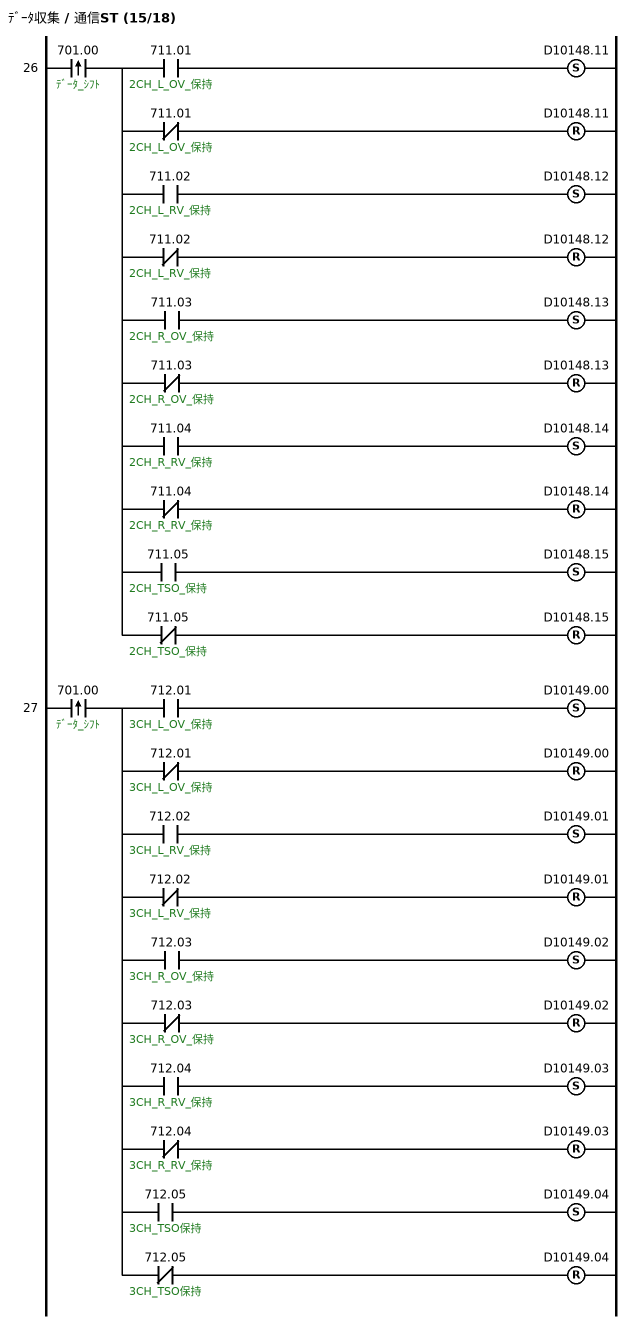
; [picture p216: ﾃﾞｰﾀ収集 / 通信ST, rungs 26-27]
; rung 26
@LD 701.00  ; ﾃﾞｰﾀ_ｼﾌﾄ
OUT TR0
AND 711.01  ; 2CH_L_OV_保持
SET D10148.11
LD TR0
ANDNOT 711.01  ; 2CH_L_OV_保持
RSET D10148.11
LD TR0
AND 711.02  ; 2CH_L_RV_保持
SET D10148.12
LD TR0
ANDNOT 711.02  ; 2CH_L_RV_保持
RSET D10148.12
LD TR0
AND 711.03  ; 2CH_R_OV_保持
SET D10148.13
LD TR0
ANDNOT 711.03  ; 2CH_R_OV_保持
RSET D10148.13
LD TR0
AND 711.04  ; 2CH_R_RV_保持
SET D10148.14
LD TR0
ANDNOT 711.04  ; 2CH_R_RV_保持
RSET D10148.14
LD TR0
AND 711.05  ; 2CH_TSO_保持
SET D10148.15
LD TR0
ANDNOT 711.05  ; 2CH_TSO_保持
RSET D10148.15
; rung 27
@LD 701.00  ; ﾃﾞｰﾀ_ｼﾌﾄ
OUT TR0
AND 712.01  ; 3CH_L_OV_保持
SET D10149.00
LD TR0
ANDNOT 712.01  ; 3CH_L_OV_保持
RSET D10149.00
LD TR0
AND 712.02  ; 3CH_L_RV_保持
SET D10149.01
LD TR0
ANDNOT 712.02  ; 3CH_L_RV_保持
RSET D10149.01
LD TR0
AND 712.03  ; 3CH_R_OV_保持
SET D10149.02
LD TR0
ANDNOT 712.03  ; 3CH_R_OV_保持
RSET D10149.02
LD TR0
AND 712.04  ; 3CH_R_RV_保持
SET D10149.03
LD TR0
ANDNOT 712.04  ; 3CH_R_RV_保持
RSET D10149.03
LD TR0
AND 712.05  ; 3CH_TSO保持
SET D10149.04
LD TR0
ANDNOT 712.05  ; 3CH_TSO保持
RSET D10149.04

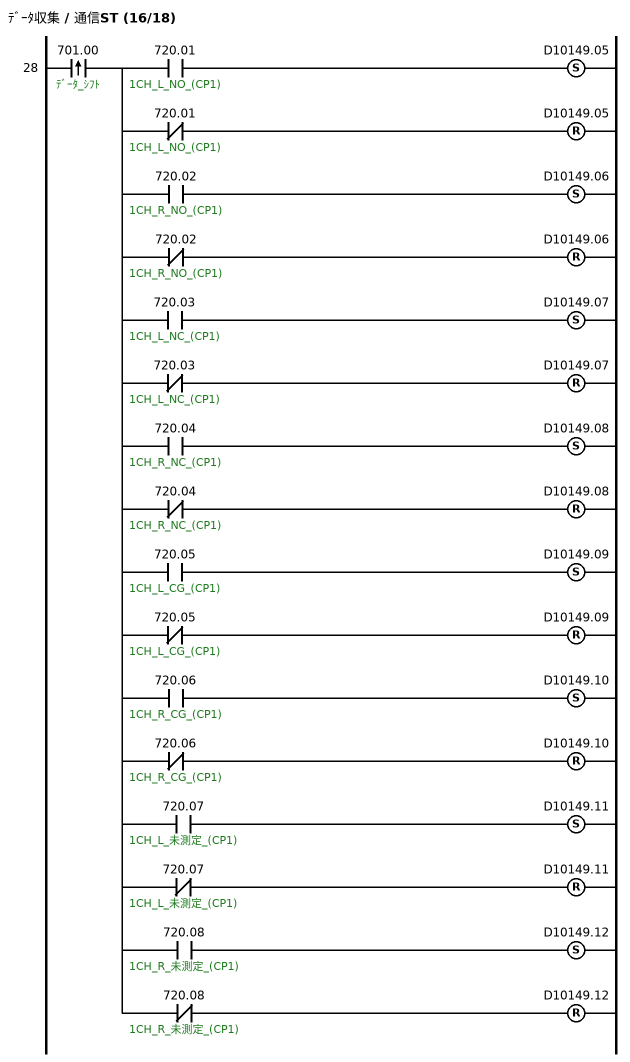
; rung 28
@LD 701.00  ; ﾃﾞｰﾀ_ｼﾌﾄ
OUT TR0
AND 720.01  ; 1CH_L_NO_(CP1)
SET D10149.05
LD TR0
ANDNOT 720.01  ; 1CH_L_NO_(CP1)
RSET D10149.05
LD TR0
AND 720.02  ; 1CH_R_NO_(CP1)
SET D10149.06
LD TR0
ANDNOT 720.02  ; 1CH_R_NO_(CP1)
RSET D10149.06
LD TR0
AND 720.03  ; 1CH_L_NC_(CP1)
SET D10149.07
LD TR0
ANDNOT 720.03  ; 1CH_L_NC_(CP1)
RSET D10149.07
LD TR0
AND 720.04  ; 1CH_R_NC_(CP1)
SET D10149.08
LD TR0
ANDNOT 720.04  ; 1CH_R_NC_(CP1)
RSET D10149.08
LD TR0
AND 720.05  ; 1CH_L_CG_(CP1)
SET D10149.09
LD TR0
ANDNOT 720.05  ; 1CH_L_CG_(CP1)
RSET D10149.09
LD TR0
AND 720.06  ; 1CH_R_CG_(CP1)
SET D10149.10
LD TR0
ANDNOT 720.06  ; 1CH_R_CG_(CP1)
RSET D10149.10
LD TR0
AND 720.07  ; 1CH_L_未測定_(CP1)
SET D10149.11
LD TR0
ANDNOT 720.07  ; 1CH_L_未測定_(CP1)
RSET D10149.11
LD TR0
AND 720.08  ; 1CH_R_未測定_(CP1)
SET D10149.12
LD TR0
ANDNOT 720.08  ; 1CH_R_未測定_(CP1)
RSET D10149.12

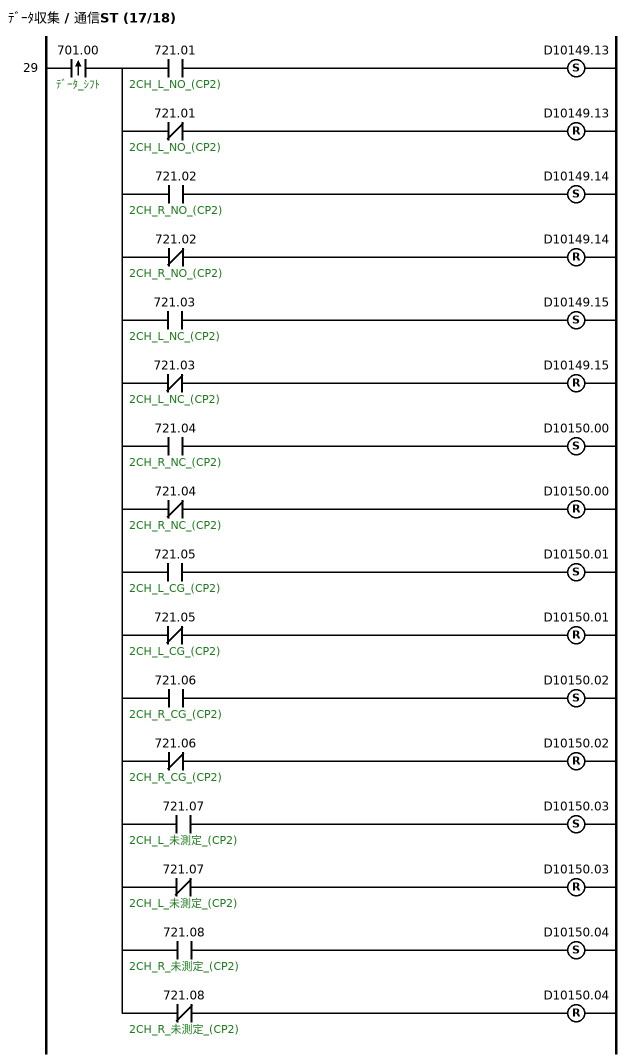
; rung 29
@LD 701.00  ; ﾃﾞｰﾀ_ｼﾌﾄ
OUT TR0
AND 721.01  ; 2CH_L_NO_(CP2)
SET D10149.13
LD TR0
ANDNOT 721.01  ; 2CH_L_NO_(CP2)
RSET D10149.13
LD TR0
AND 721.02  ; 2CH_R_NO_(CP2)
SET D10149.14
LD TR0
ANDNOT 721.02  ; 2CH_R_NO_(CP2)
RSET D10149.14
LD TR0
AND 721.03  ; 2CH_L_NC_(CP2)
SET D10149.15
LD TR0
ANDNOT 721.03  ; 2CH_L_NC_(CP2)
RSET D10149.15
LD TR0
AND 721.04  ; 2CH_R_NC_(CP2)
SET D10150.00
LD TR0
ANDNOT 721.04  ; 2CH_R_NC_(CP2)
RSET D10150.00
LD TR0
AND 721.05  ; 2CH_L_CG_(CP2)
SET D10150.01
LD TR0
ANDNOT 721.05  ; 2CH_L_CG_(CP2)
RSET D10150.01
LD TR0
AND 721.06  ; 2CH_R_CG_(CP2)
SET D10150.02
LD TR0
ANDNOT 721.06  ; 2CH_R_CG_(CP2)
RSET D10150.02
LD TR0
AND 721.07  ; 2CH_L_未測定_(CP2)
SET D10150.03
LD TR0
ANDNOT 721.07  ; 2CH_L_未測定_(CP2)
RSET D10150.03
LD TR0
AND 721.08  ; 2CH_R_未測定_(CP2)
SET D10150.04
LD TR0
ANDNOT 721.08  ; 2CH_R_未測定_(CP2)
RSET D10150.04

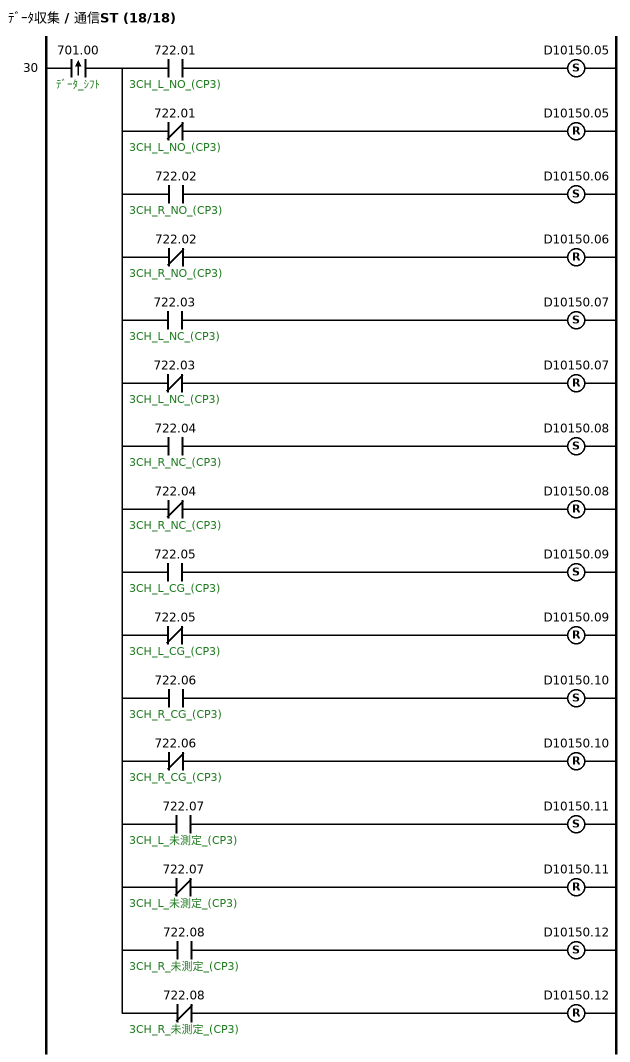
; rung 30
@LD 701.00  ; ﾃﾞｰﾀ_ｼﾌﾄ
OUT TR0
AND 722.01  ; 3CH_L_NO_(CP3)
SET D10150.05
LD TR0
ANDNOT 722.01  ; 3CH_L_NO_(CP3)
RSET D10150.05
LD TR0
AND 722.02  ; 3CH_R_NO_(CP3)
SET D10150.06
LD TR0
ANDNOT 722.02  ; 3CH_R_NO_(CP3)
RSET D10150.06
LD TR0
AND 722.03  ; 3CH_L_NC_(CP3)
SET D10150.07
LD TR0
ANDNOT 722.03  ; 3CH_L_NC_(CP3)
RSET D10150.07
LD TR0
AND 722.04  ; 3CH_R_NC_(CP3)
SET D10150.08
LD TR0
ANDNOT 722.04  ; 3CH_R_NC_(CP3)
RSET D10150.08
LD TR0
AND 722.05  ; 3CH_L_CG_(CP3)
SET D10150.09
LD TR0
ANDNOT 722.05  ; 3CH_L_CG_(CP3)
RSET D10150.09
LD TR0
AND 722.06  ; 3CH_R_CG_(CP3)
SET D10150.10
LD TR0
ANDNOT 722.06  ; 3CH_R_CG_(CP3)
RSET D10150.10
LD TR0
AND 722.07  ; 3CH_L_未測定_(CP3)
SET D10150.11
LD TR0
ANDNOT 722.07  ; 3CH_L_未測定_(CP3)
RSET D10150.11
LD TR0
AND 722.08  ; 3CH_R_未測定_(CP3)
SET D10150.12
LD TR0
ANDNOT 722.08  ; 3CH_R_未測定_(CP3)
RSET D10150.12

### Section END
; rung 0
END(001)